FUNCTION_BLOCK Station001 EXTENDS TcoCore.TcoContext
VAR
	_sequence : Station001_Sequencer(THIS^, FALSE);
END_VAR

(*~
	<docu>
		<summary>
			Main method of the TcoContext. This is the entry point of any control logic that belongs to this context. 
			The call of this method is ensured by calling the <c>InstanceName.Run()</c> method, and it must not be called explicitly.
			This method is abstract, and it must be overridden in derived block.
		</summary>
	</docu>
~*)
METHOD PROTECTED  Main
_sequence.Run();
END_METHOD

END_FUNCTION_BLOCK

(* stored: Version 1.1.0.1, ProductVersion 3.1.4024.6
   POU Station001: Id {00a3bb22-82f5-4ea8-82e2-290ee3363eb4}, SpecialFunc None
   Method Main: Id {e83e3098-35a6-4623-baf3-b3eac487355d} *)
